FUNCTION Init_PB_Mom_75x75 : INT

VAR_INPUT
END_VAR

VAR

END_VAR

VAR_IN_OUT
	COMP:TS_Component;
END_VAR

COMP.B_TYPE:=0;
COMP.size:=1;

END_FUNCTION

(* stored: Version 1.1.0.1, ProductVersion 3.1.4020.12
   POU Init_PB_Mom_75x75: Id {b4edcf78-53a3-478a-a60c-a863f7075b5a}, SpecialFunc None *)
